PROGRAM CanReceiver
VAR
	fbUdp1 : FB_CanReceiver;
END_VAR

fbUdp1();

END_PROGRAM

(* stored: Version 1.1.0.1, ProductVersion 3.1.4024.12
   POU CanReceiver: Id {b267492c-8f20-4396-8f9a-bf5860142b18}, SpecialFunc None *)
